// Mitsubishi GX Works2 project: yudomotor   PLC: Q03UDV

PROGRAM MAIN
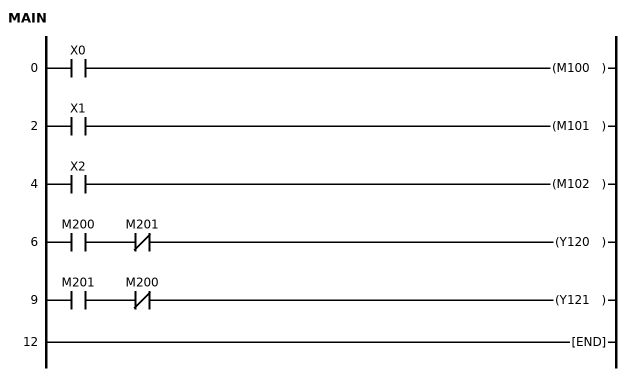
0     LD      X0
      OUT     M100
2     LD      X1
      OUT     M101
4     LD      X2
      OUT     M102
6     LD      M200
      ANI     M201
      OUT     Y120
9     LD      M201
      ANI     M200
      OUT     Y121
12    END
END_PROGRAM
